FUNCTION_BLOCK EL1124
VAR
	_io : EL1xx4_Data;
	{attribute addProperty Name "WcState"}
	_wcState : WcStateInputToggle;
	{attribute addProperty Name "Info data"}
	_infoData : InfoDataBase;
END_VAR

PROPERTY IO : REFERENCE TO EL1xx4_Data
GET
IO REF= _io;
END_GET
END_PROPERTY

PROPERTY WcState : REFERENCE TO WcStateInputToggle
GET
WcState REF= _wcState;
END_GET
END_PROPERTY

END_FUNCTION_BLOCK

(* stored: Version 1.1.0.1, ProductVersion 3.1.4024.9
   POU EL1124: Id {7c981941-76ed-0d45-07f5-3ba6da52ca5b}, SpecialFunc None
   Property IO: Id {aed10be0-187c-0de4-2c13-90d6a16fe0ec}
   Get Get: Id {655998a4-cac5-0dce-2f94-8479d917dcaa}
   Property WcState: Id {8a03c858-b7bf-02e8-2b8d-003ca1b52db2}
   Get Get: Id {4d10c1e4-5a0d-0c0b-23a6-633e02e900d0} *)
